// Mitsubishi GX Works2 project: 240920_공급가공실린더   PLC: Q03UDV

PROGRAM SUB
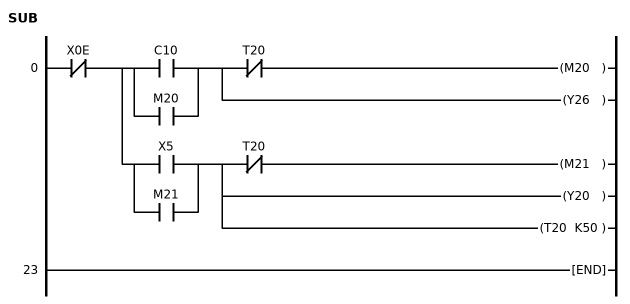
0     LDI     X0E
      MPS
      LD      C10
      OR      M20
      ANB
      MPS
      ANI     T20
      OUT     M20
      MPP
      OUT     Y26
      MPP
      LD      X5
      OR      M21
      ANB
      MPS
      ANI     T20
      OUT     M21
      MPP
      OUT     Y20
      OUT     T20 K50
23    END
END_PROGRAM

PROGRAM MAIN
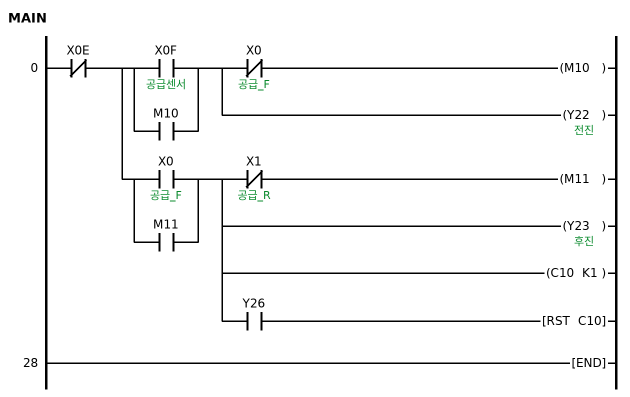
0     LDI     X0E
      MPS
      LD      X0F  ; 공급센서
      OR      M10
      ANB
      MPS
      ANI     X0  ; 공급_F
      OUT     M10
      MPP
      OUT     Y22  ; 전진
      MPP
      LD      X0  ; 공급_F
      OR      M11
      ANB
      MPS
      ANI     X1  ; 공급_R
      OUT     M11
      MPP
      OUT     Y23  ; 후진
      OUT     C10 K1
      AND     Y26
      RST     C10
28    END
END_PROGRAM
